// Mitsubishi GX Works2 project: PLC_GROUP_15   PLC: FX3G

// global labels: Global1
VAR_GLOBAL
  Start_Day AT X007 : BOOL;
  End_Day AT M5 : BOOL;
  Work_Day_On AT Y007 : BOOL;
  Input_Raspberry AT D1100 : REAL;
  Input_Lemon AT D1104 : REAL;
  Input_Stabilizer AT D1108 : REAL;
  Input_Gummy AT D1112 : REAL;
  Raspberry_Amount AT D1102 : REAL;
  Lemon_Amount AT D1106 : REAL;
  Stabilizer_Amount AT D1110 : REAL;
  Gummy_Amount AT D1114 : REAL;
  Close_Reset_1 AT CS0 : BOOL;
  Package_Container AT D1126 : REAL;
END_VAR
VAR_GLOBAL CONSTANT
  To_Esroni : REAL := 40;  (* 40 *)
END_VAR
VAR_GLOBAL
  Analog_Output AT D8282 : REAL;
  One_Time_Reset AT CC0 : BOOL;
  Start_Production AT X001 : BOOL;
  Save_Analog_Value AT D8201 : REAL;
END_VAR
VAR_GLOBAL CONSTANT
  CONST400 : REAL := 400;  (* 400 *)
  Min_Regular : REAL;  (* 0 *)
  Max_Regular : REAL := 5;  (* 5 *)
  Min_Pinook : REAL := 6;  (* 6 *)
  Max_Pinook : REAL := 10;  (* 10 *)
END_VAR
VAR_GLOBAL
  Regular AT M3 : BOOL;
  Pinook AT M4 : BOOL;
END_VAR
VAR_GLOBAL CONSTANT
  Check1 : INT := 1;  (* 1 *)
END_VAR
VAR_GLOBAL
  Analog_Input_1 AT D8280 : INT;
  Analog_Real_Value AT D1128 : REAL;
END_VAR
VAR_GLOBAL CONSTANT
  Min_Raspberry_Regular : REAL := 280;  (* 280 *)
  Min_Raspberry_Pinook : REAL := 385;  (* 385 *)
  Min_Lemon_Regular : REAL := 455;  (* 455 *)
  Min_Lemon_Pinook : REAL := 665;  (* 665 *)
  Min_Stabilizer_Regular : REAL := 105;  (* 105 *)
  Min_Stabilizer_Pinook : REAL := 210;  (* 210 *)
  Min_Gummy_Regular : REAL := 28;  (* 28 *)
  Min_Gummy_Pinook : REAL := 70;  (* 70 *)
END_VAR
VAR_GLOBAL
  Check_Product_Raspberry AT M10 : BOOL;
  Check_Product_Lemon AT M20 : BOOL;
  Check_Product_Stabilizer AT M30 : BOOL;
  Check_Product_Gummy AT M40 : BOOL;
  Enough_Products AT M1 : BOOL;
  No_Inventory AT M6 : BOOL;
  Emergency AT X005 : BOOL;
  Timer1 AT TC1 : BOOL;
END_VAR
VAR_GLOBAL CONSTANT
  CONST_5Sec : WORD := 50;  (* 50 *)
END_VAR
VAR_GLOBAL
  Timer_1_Finish AT TS1 : BOOL;
  FiveSecLight AT Y000 : BOOL;
END_VAR
VAR_GLOBAL CONSTANT
  SUB_Res_K280 : REAL := 280;  (* 280 *)
  SUB_Lemon_K455 : REAL := 455;  (* 455 *)
  SUB_Stabi_K105 : REAL := 105;  (* 105 *)
  ADD_Stabi_K35 : REAL := 35;  (* 35 *)
  ADD_Lemon_K455 : REAL := 455;  (* 455 *)
  ADD_Res_K280 : REAL := 280;  (* 280 *)
  ADD_Stabi_K70 : REAL := 70;  (* 70 *)
END_VAR
VAR_GLOBAL
  Raspberry_Cooling_Container AT D1120 : REAL;
  Lemon_Making_Container AT D1118 : REAL;
  Raspberry_Making_Container AT D1116 : REAL;
END_VAR
VAR_GLOBAL CONSTANT
  CONST0 : REAL;  (* 0 *)
  SUB_Res_K385 : REAL := 385;  (* 385 *)
  SUB_Lemon_K665 : REAL := 665;  (* 665 *)
  SUB_Stabi_K210 : REAL := 210;  (* 210 *)
  ADD_Res_K385 : REAL := 385;  (* 385 *)
  ADD_Lemon_K665 : REAL := 665;  (* 665 *)
  ADD_Stabi_K140 : REAL := 140;  (* 140 *)
END_VAR
VAR_GLOBAL
  Can_Start_Cooling AT M21 : BOOL;
  Start_Cooling AT X002 : BOOL;
  Making_finish AT M22 : BOOL;
  Counter_2_finish AT TS2 : BOOL;
  Temperature AT X003 : BOOL;
  CoolingLight AT Y002 : BOOL;
  Timer2 AT TC2 : BOOL;
END_VAR
VAR_GLOBAL CONSTANT
  CONST_8Sec : INT := 80;  (* 80 *)
END_VAR
VAR_GLOBAL
  Lemon_Cooling_Container AT D1122 : REAL;
  Cooling_Finish AT M23 : BOOL;
  Temperature_On AT M24 : BOOL;
END_VAR
VAR_GLOBAL CONSTANT
  SUB_Gummy_K28 : REAL := 28;  (* 28 *)
  SUB_Gummy_K70 : REAL := 70;  (* 70 *)
  ADD_Gummy_K70 : REAL := 70;  (* 70 *)
  ADD_Gummy_K28 : REAL := 28;  (* 28 *)
END_VAR
VAR_GLOBAL
  Mixing_Container AT D1124 : REAL;
  Twinkle_Stop AT M41 : BOOL;
  M_0 AT M0 : BOOL;
  Counter_3_finish AT TS3 : BOOL;
  Timer3 AT TC3 : BOOL;
END_VAR
VAR_GLOBAL CONSTANT
  CONST_1Sec : INT := 10;
END_VAR
VAR_GLOBAL
  Timer4 AT TC4 : BOOL;
  Counter_4_finish AT TS4 : BOOL;  (* 10 *)
  Y_6 AT Y006 : BOOL;
  Y_5 AT Y005 : BOOL;
  Timer5 AT TC5 : BOOL;
END_VAR
VAR_GLOBAL CONSTANT
  Pinook_Blend_Time : INT := 50;  (* 50 *)
  Regular_Blend_Time : INT := 30;  (* 30 *)
END_VAR
VAR_GLOBAL
  Timer6 AT TC6 : BOOL;
  Counter_5_finish AT TS5 : BOOL;
  Counter_6_finish AT TS6 : BOOL;
  Packing_Begin AT M42 : BOOL;
END_VAR
VAR_GLOBAL CONSTANT
  ADD_1_Package : REAL := 1;  (* 1 *)
END_VAR
VAR_GLOBAL
  Cycle_Finished AT M44 : BOOL;
  Timer_3_finish AT TS3 : BOOL;
  Timer_4_finish AT TS4 : BOOL;  (* 10 *)
  Timer_5_finish AT TS5 : BOOL;
  Timer_6_finish AT TS6 : BOOL;
  Timer_2_finish AT TS2 : BOOL;
END_VAR

// task Task_01 (event TRUE, interval 0, priority 31): POU_01

PROGRAM POU_01
(* structured ladder/FBD written out as ST: instructions are called as NAME(EN, inputs, outputs); _pN, _eN, _tN stand for wires *)
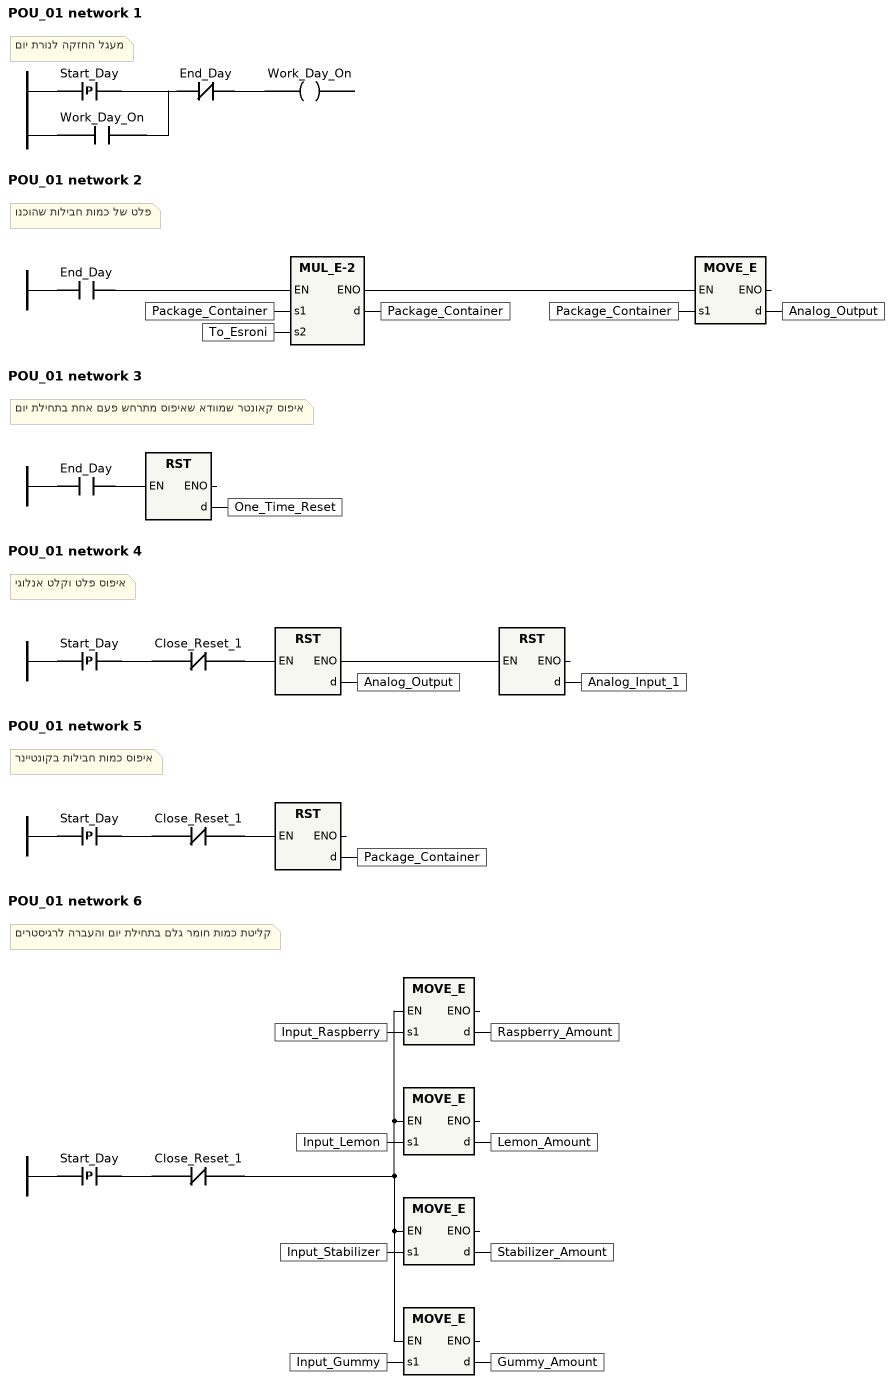
(* network 1 *)
(* מעגל החזקה לנורת יום *)
Work_Day_On := (LDP(TRUE, Start_Day) OR Work_Day_On) AND NOT End_Day;
(* network 2 *)
(* פלט של כמות חבילות שהוכנו *)
_e1 := MUL_E(End_Day, Package_Container, To_Esroni, Package_Container);
MOVE_E(_e1, Package_Container, Analog_Output);
(* network 3 *)
(* איפוס קאונטר שמוודא שאיפוס מתרחש פעם אחת בתחילת יום *)
RST(End_Day, One_Time_Reset);
(* network 4 *)
(* איפוס פלט וקלט אנלוגי *)
_e1 := RST(LDP(TRUE, Start_Day) AND NOT Close_Reset_1, Analog_Output);
RST(_e1, Analog_Input_1);
(* network 5 *)
(* איפוס כמות חבילות בקונטיינר *)
RST(LDP(TRUE, Start_Day) AND NOT Close_Reset_1, Package_Container);
(* network 6 *)
(* קליטת כמות חומר גלם בתחילת יום והעברה לרגיסטרים *)
_p1 := LDP(TRUE, Start_Day) AND NOT Close_Reset_1;
MOVE_E(_p1, Input_Raspberry, Raspberry_Amount);
MOVE_E(_p1, Input_Lemon, Lemon_Amount);
MOVE_E(_p1, Input_Stabilizer, Stabilizer_Amount);
MOVE_E(_p1, Input_Gummy, Gummy_Amount);
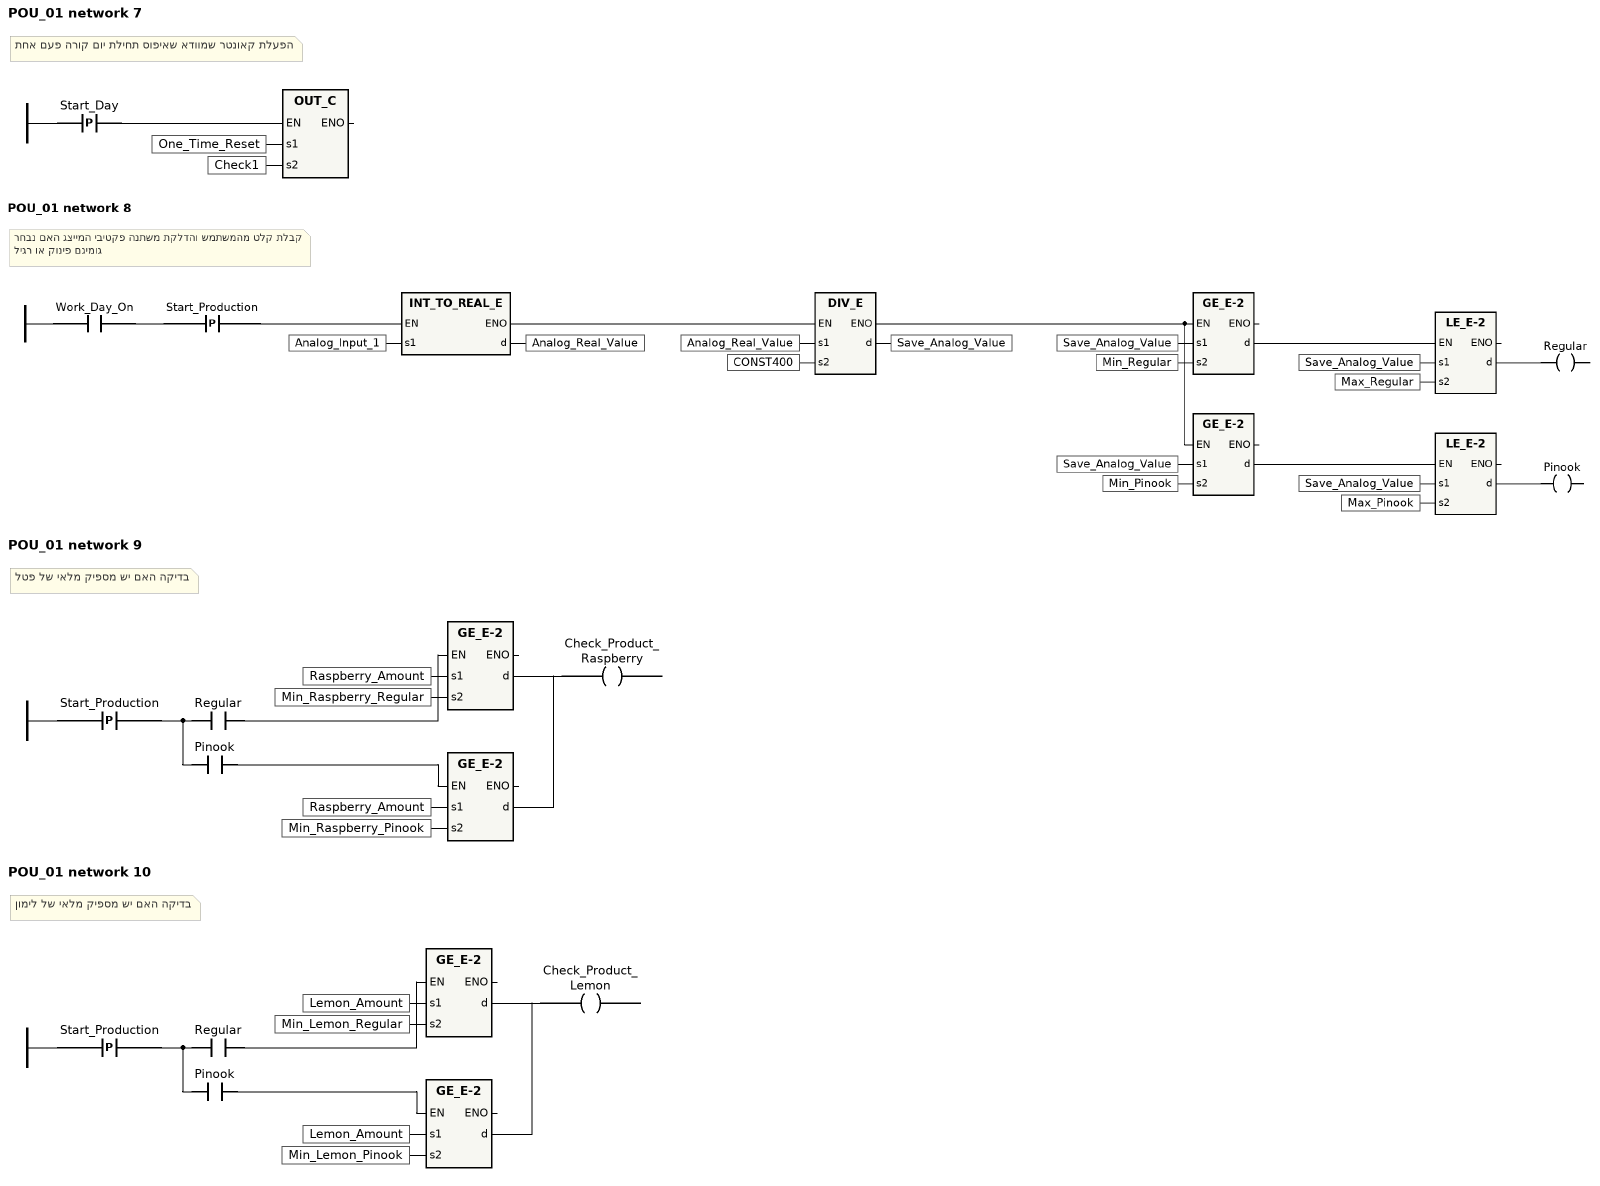
(* network 7 *)
(* הפעלת קאונטר שמוודא שאיפוס תחילת יום קורה פעם אחת *)
OUT_C(LDP(TRUE, Start_Day), One_Time_Reset, Check1);
(* network 8 *)
(* קבלת קלט מהמשתמש והדלקת משתנה פקטיבי המייצג האם נבחר גומיגם פינוק או רגיל *)
_e1 := INT_TO_REAL_E(Work_Day_On AND LDP(TRUE, Start_Production), Analog_Input_1, Analog_Real_Value);
_e2 := DIV_E(_e1, Analog_Real_Value, CONST400, Save_Analog_Value);
GE_E(_e2, Save_Analog_Value, Min_Regular, _t3);
LE_E(_t3, Save_Analog_Value, Max_Regular, _t4);
Regular := _t4;
GE_E(_e2, Save_Analog_Value, Min_Pinook, _t5);
LE_E(_t5, Save_Analog_Value, Max_Pinook, _t6);
Pinook := _t6;
(* network 9 *)
(* בדיקה האם יש מספיק מלאי של פטל *)
_p1 := LDP(TRUE, Start_Production);
GE_E(_p1 AND Regular, Raspberry_Amount, Min_Raspberry_Regular, _t2);
GE_E(_p1 AND Pinook, Raspberry_Amount, Min_Raspberry_Pinook, _t3);
Check_Product_Raspberry := _t2 OR _t3;
(* network 10 *)
(* בדיקה האם יש מספיק מלאי של לימון *)
_p1 := LDP(TRUE, Start_Production);
GE_E(_p1 AND Regular, Lemon_Amount, Min_Lemon_Regular, _t2);
GE_E(_p1 AND Pinook, Lemon_Amount, Min_Lemon_Pinook, _t3);
Check_Product_Lemon := _t2 OR _t3;
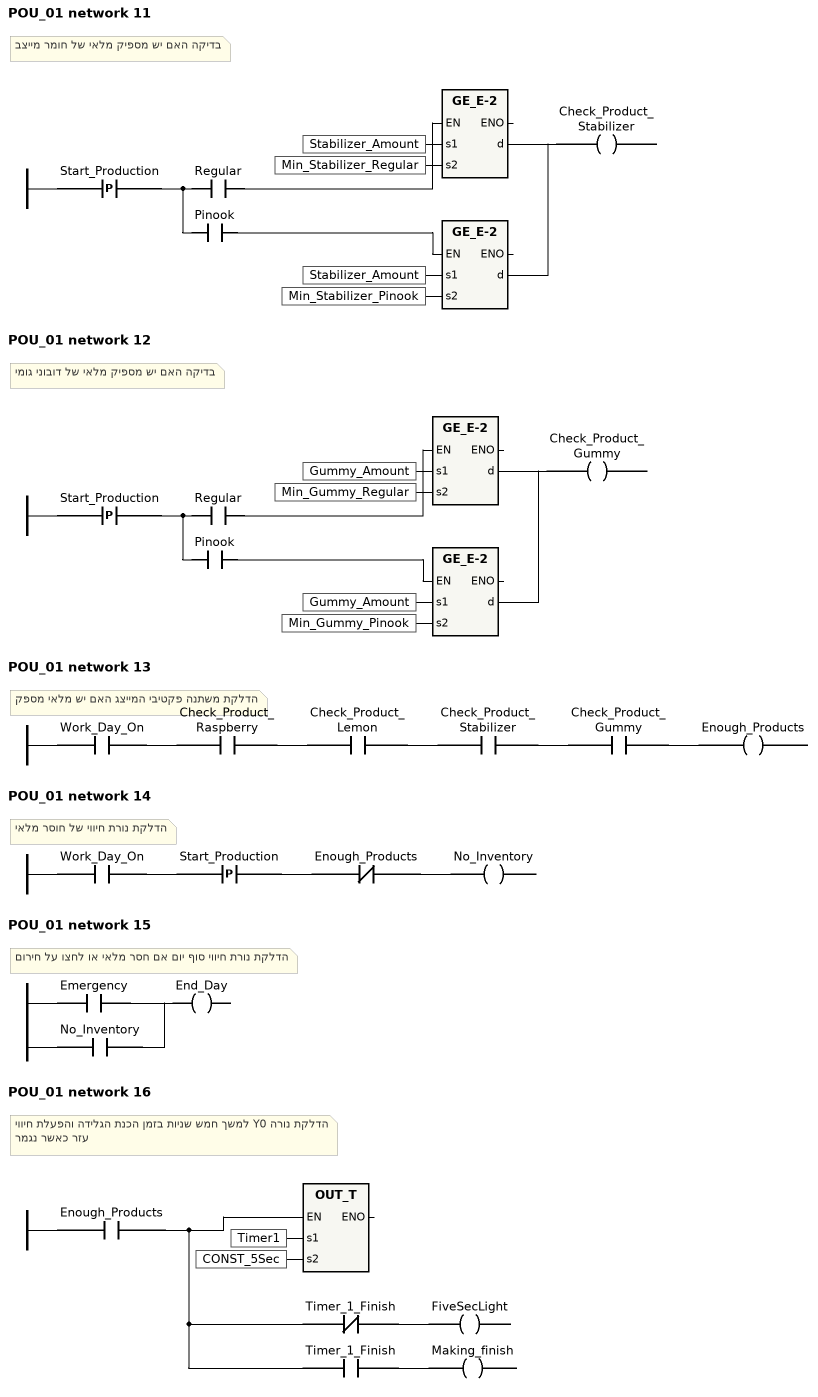
(* network 11 *)
(* בדיקה האם יש מספיק מלאי של חומר מייצב *)
_p1 := LDP(TRUE, Start_Production);
GE_E(_p1 AND Regular, Stabilizer_Amount, Min_Stabilizer_Regular, _t2);
GE_E(_p1 AND Pinook, Stabilizer_Amount, Min_Stabilizer_Pinook, _t3);
Check_Product_Stabilizer := _t2 OR _t3;
(* network 12 *)
(* בדיקה האם יש מספיק מלאי של דובוני גומי *)
_p1 := LDP(TRUE, Start_Production);
GE_E(_p1 AND Regular, Gummy_Amount, Min_Gummy_Regular, _t2);
GE_E(_p1 AND Pinook, Gummy_Amount, Min_Gummy_Pinook, _t3);
Check_Product_Gummy := _t2 OR _t3;
(* network 13 *)
(* הדלקת משתנה פקטיבי המייצג האם יש מלאי מספק *)
Enough_Products := Work_Day_On AND Check_Product_Raspberry AND Check_Product_Lemon AND Check_Product_Stabilizer AND Check_Product_Gummy;
(* network 14 *)
(* הדלקת נורת חיווי של חוסר מלאי *)
No_Inventory := Work_Day_On AND LDP(TRUE, Start_Production) AND NOT Enough_Products;
(* network 15 *)
(* הדלקת נורת חיווי סוף יום אם חסר מלאי או לחצו על חירום *)
End_Day := Emergency OR No_Inventory;
(* network 16 *)
(* הדלקת נורה Y0 למשך חמש שניות בזמן הכנת הגלידה והפעלת חיווי עזר כאשר נגמר *)
FiveSecLight := Enough_Products AND NOT Timer_1_Finish;
OUT_T(Enough_Products, Timer1, CONST_5Sec);
Making_finish := Enough_Products AND Timer_1_Finish;
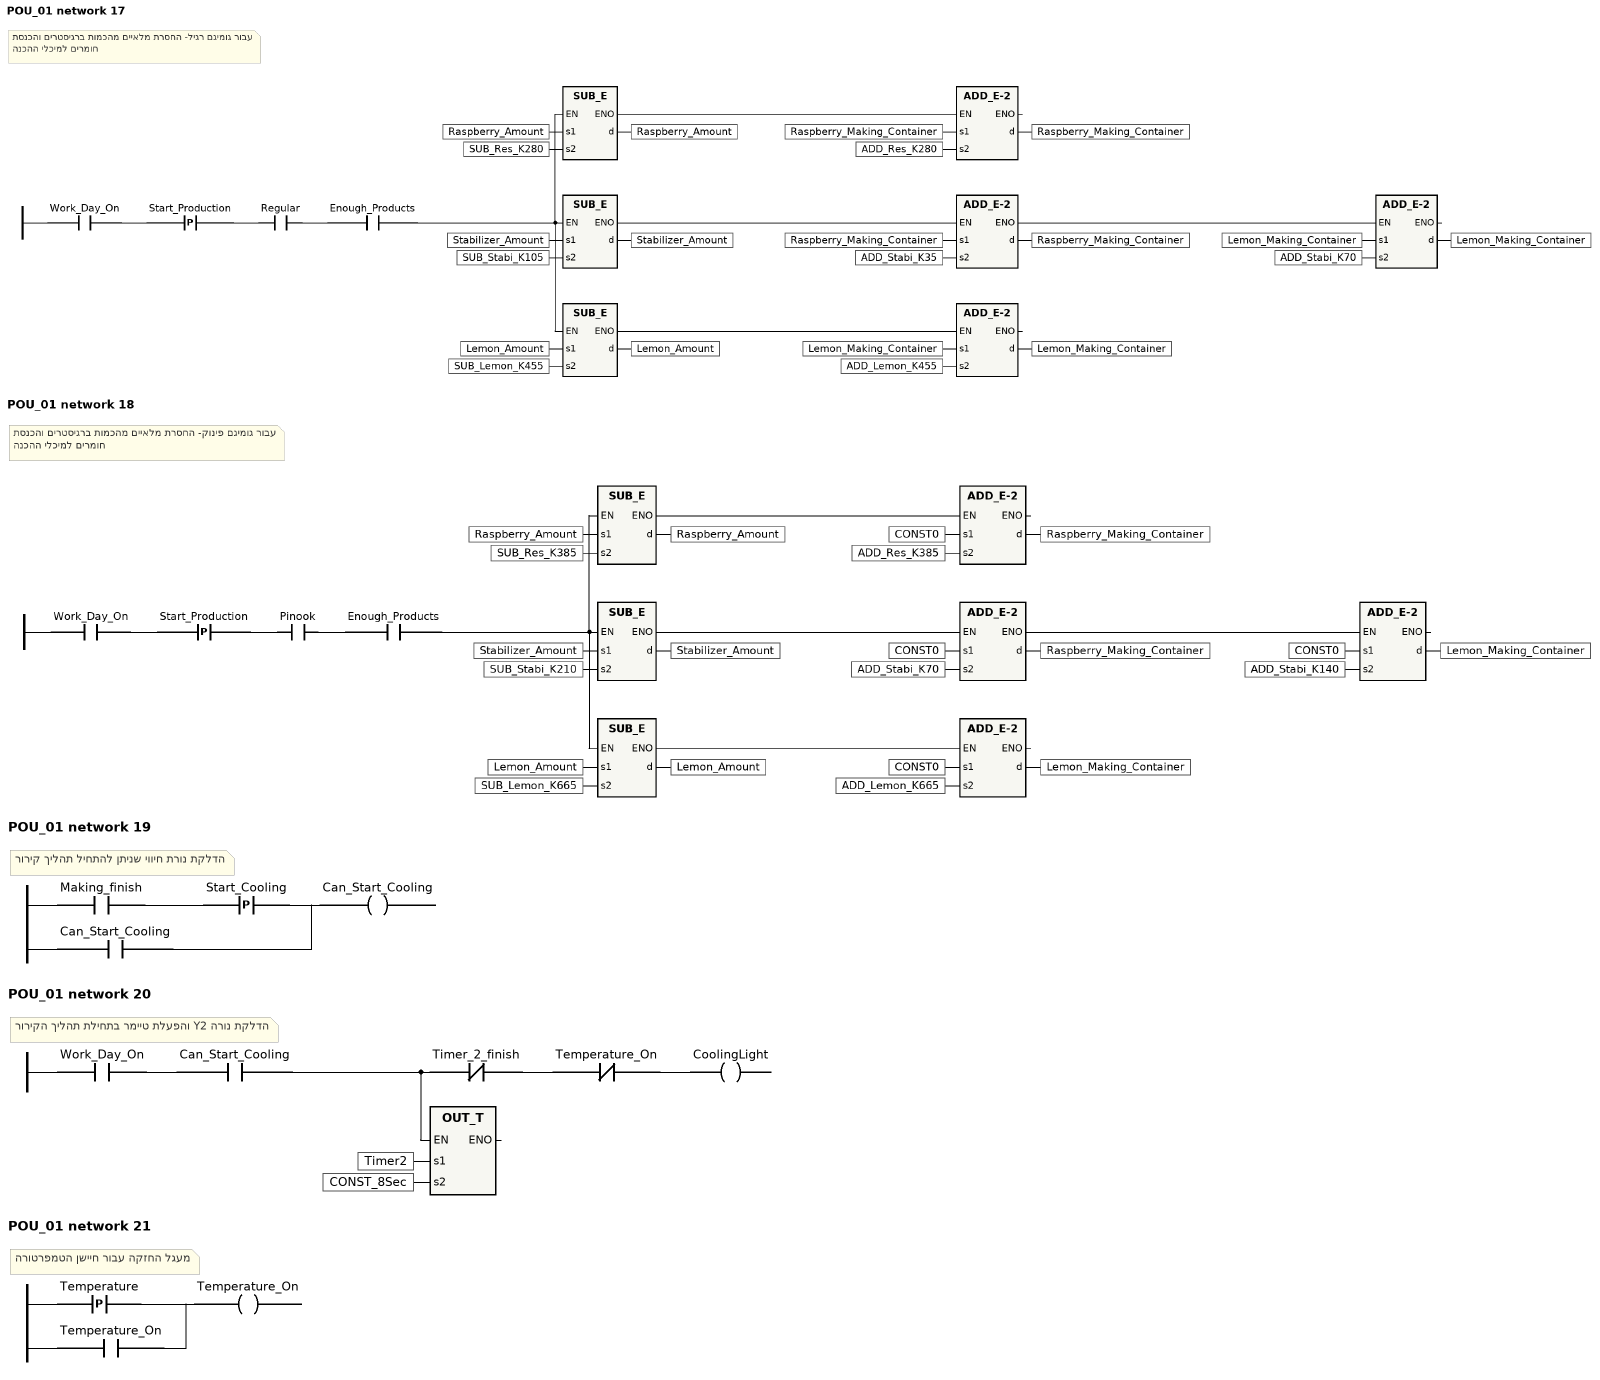
(* network 17 *)
(* עבור גומיגם רגיל- החסרת מלאיים מהכמות ברגיסטרים והכנסת חומרים למיכלי ההכנה *)
_p1 := Work_Day_On AND LDP(TRUE, Start_Production) AND Regular AND Enough_Products;
_e2 := SUB_E(_p1, Raspberry_Amount, SUB_Res_K280, Raspberry_Amount);
ADD_E(_e2, Raspberry_Making_Container, ADD_Res_K280, Raspberry_Making_Container);
_e3 := SUB_E(_p1, Lemon_Amount, SUB_Lemon_K455, Lemon_Amount);
ADD_E(_e3, Lemon_Making_Container, ADD_Lemon_K455, Lemon_Making_Container);
_e4 := SUB_E(_p1, Stabilizer_Amount, SUB_Stabi_K105, Stabilizer_Amount);
_e5 := ADD_E(_e4, Raspberry_Making_Container, ADD_Stabi_K35, Raspberry_Making_Container);
ADD_E(_e5, Lemon_Making_Container, ADD_Stabi_K70, Lemon_Making_Container);
(* network 18 *)
(* עבור גומיגם פינוק- החסרת מלאיים מהכמות ברגיסטרים והכנסת חומרים למיכלי ההכנה *)
_p1 := Work_Day_On AND LDP(TRUE, Start_Production) AND Pinook AND Enough_Products;
_e2 := SUB_E(_p1, Raspberry_Amount, SUB_Res_K385, Raspberry_Amount);
ADD_E(_e2, CONST0, ADD_Res_K385, Raspberry_Making_Container);
_e3 := SUB_E(_p1, Lemon_Amount, SUB_Lemon_K665, Lemon_Amount);
ADD_E(_e3, CONST0, ADD_Lemon_K665, Lemon_Making_Container);
_e4 := SUB_E(_p1, Stabilizer_Amount, SUB_Stabi_K210, Stabilizer_Amount);
_e5 := ADD_E(_e4, CONST0, ADD_Stabi_K70, Raspberry_Making_Container);
ADD_E(_e5, CONST0, ADD_Stabi_K140, Lemon_Making_Container);
(* network 19 *)
(* הדלקת נורת חיווי שניתן להתחיל תהליך קירור *)
Can_Start_Cooling := (Making_finish AND LDP(TRUE, Start_Cooling)) OR Can_Start_Cooling;
(* network 20 *)
(* הדלקת נורה Y2 והפעלת טיימר בתחילת תהליך הקירור *)
_p1 := Work_Day_On AND Can_Start_Cooling;
CoolingLight := _p1 AND NOT Timer_2_finish AND NOT Temperature_On;
OUT_T(_p1, Timer2, CONST_8Sec);
(* network 21 *)
(* מעגל החזקה עבור חיישן הטמפרטורה *)
Temperature_On := LDP(TRUE, Temperature) OR Temperature_On;
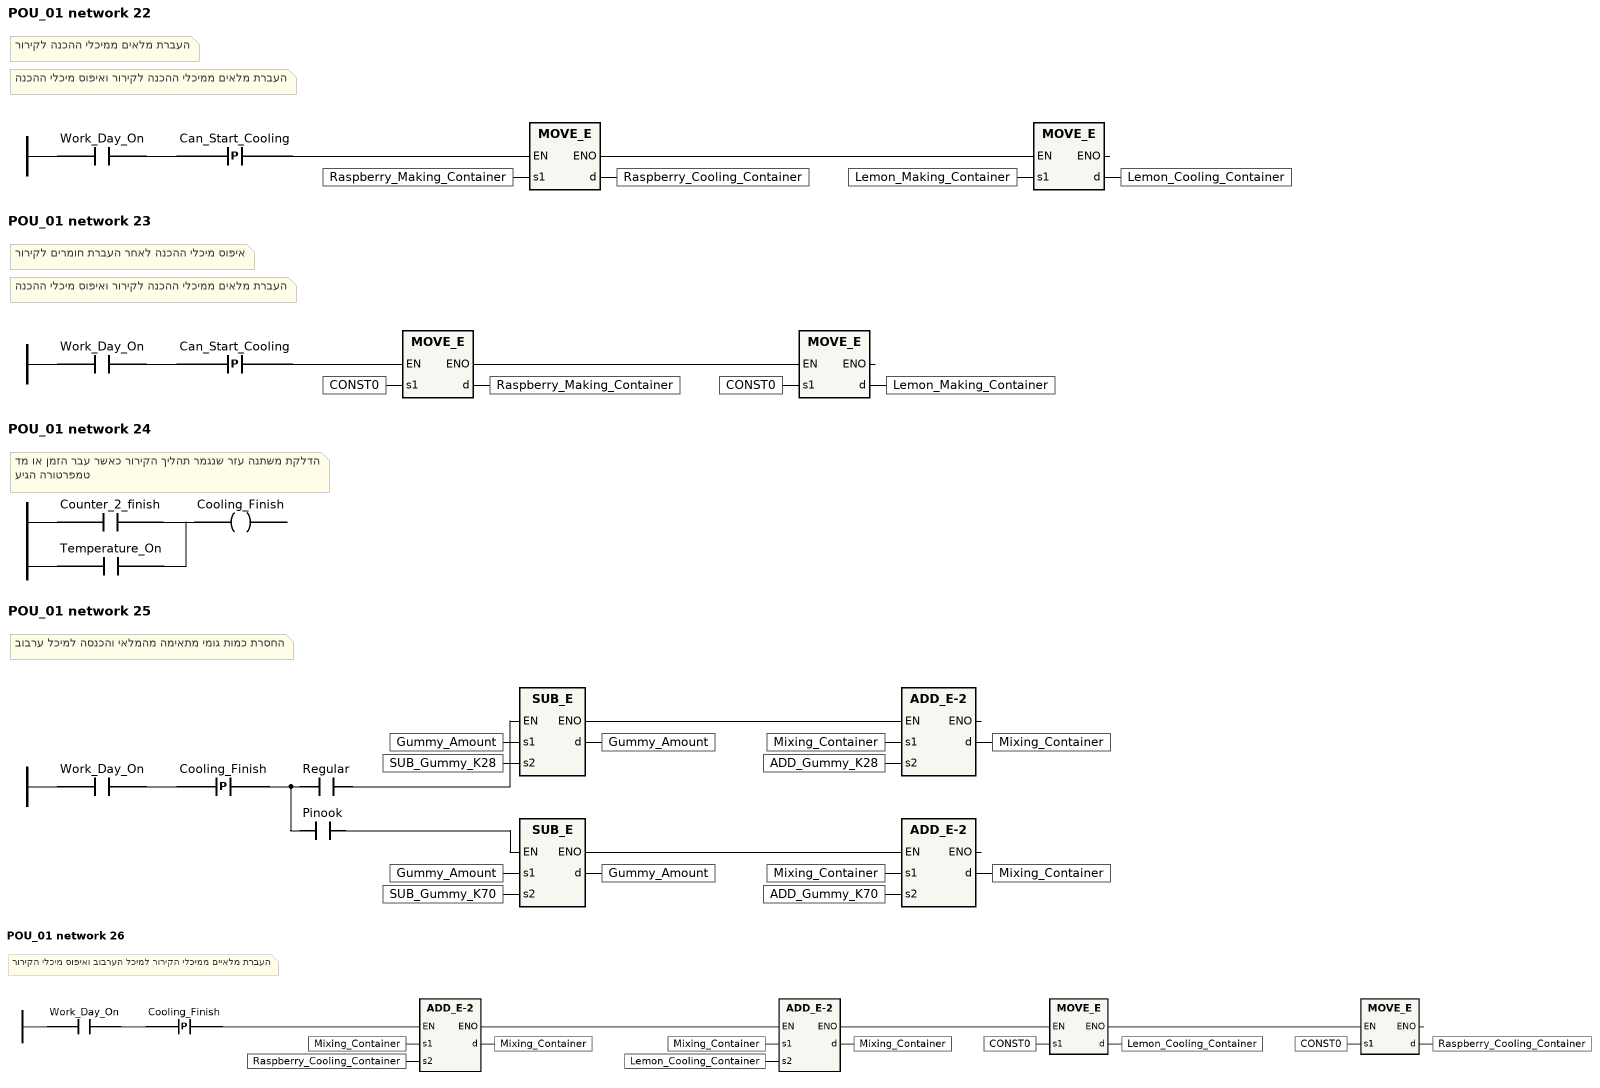
(* network 22 *)
(* העברת מלאים ממיכלי ההכנה לקירור *)
(* העברת מלאים ממיכלי ההכנה לקירור ואיפוס מיכלי ההכנה *)
_e1 := MOVE_E(Work_Day_On AND LDP(TRUE, Can_Start_Cooling), Raspberry_Making_Container, Raspberry_Cooling_Container);
MOVE_E(_e1, Lemon_Making_Container, Lemon_Cooling_Container);
(* network 23 *)
(* איפוס מיכלי ההכנה לאחר העברת חומרים לקירור *)
(* העברת מלאים ממיכלי ההכנה לקירור ואיפוס מיכלי ההכנה *)
_e1 := MOVE_E(Work_Day_On AND LDP(TRUE, Can_Start_Cooling), CONST0, Raspberry_Making_Container);
MOVE_E(_e1, CONST0, Lemon_Making_Container);
(* network 24 *)
(* הדלקת משתנה עזר שנגמר תהליך הקירור כאשר עבר הזמן או מד טמפרטורה הגיע *)
Cooling_Finish := Counter_2_finish OR Temperature_On;
(* network 25 *)
(* החסרת כמות גומי מתאימה מהמלאי והכנסה למיכל ערבוב *)
_p1 := Work_Day_On AND LDP(TRUE, Cooling_Finish);
_e2 := SUB_E(_p1 AND Regular, Gummy_Amount, SUB_Gummy_K28, Gummy_Amount);
ADD_E(_e2, Mixing_Container, ADD_Gummy_K28, Mixing_Container);
_e3 := SUB_E(_p1 AND Pinook, Gummy_Amount, SUB_Gummy_K70, Gummy_Amount);
ADD_E(_e3, Mixing_Container, ADD_Gummy_K70, Mixing_Container);
(* network 26 *)
(* העברת מלאיים ממיכלי הקירור למיכל הערבוב ואיפוס מיכלי הקירור *)
_e1 := ADD_E(Work_Day_On AND LDP(TRUE, Cooling_Finish), Mixing_Container, Raspberry_Cooling_Container, Mixing_Container);
_e2 := ADD_E(_e1, Mixing_Container, Lemon_Cooling_Container, Mixing_Container);
_e3 := MOVE_E(_e2, CONST0, Lemon_Cooling_Container);
MOVE_E(_e3, CONST0, Raspberry_Cooling_Container);
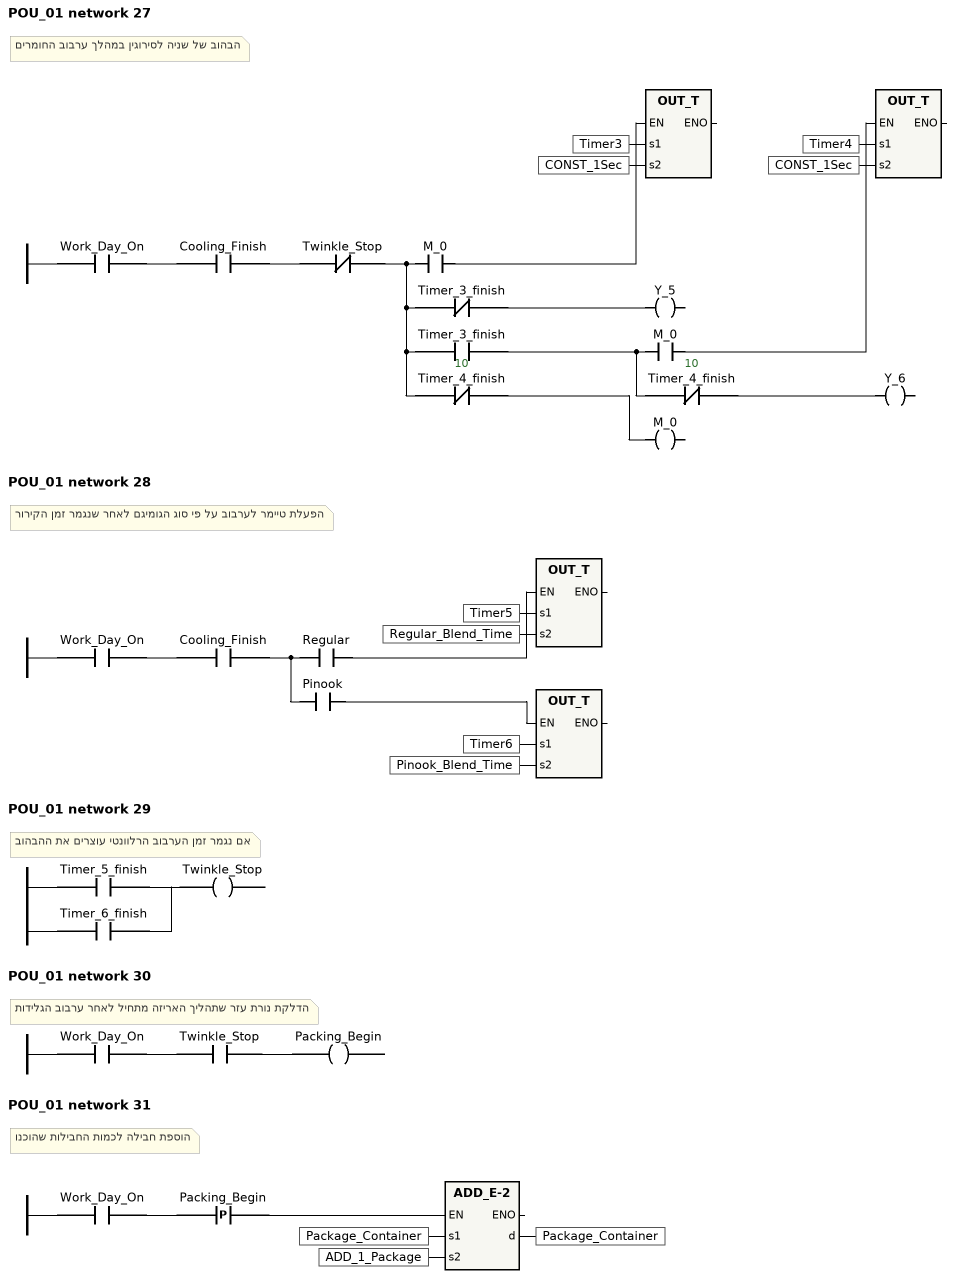
(* network 27 *)
(* הבהוב של שניה לסירוגין במהלך ערבוב החומרים *)
_p1 := Work_Day_On AND Cooling_Finish AND NOT Twinkle_Stop;
OUT_T(_p1 AND M_0, Timer3, CONST_1Sec);
Y_5 := _p1 AND NOT Timer_3_finish;
_p2 := _p1 AND Timer_3_finish;
OUT_T(_p2 AND M_0, Timer4, CONST_1Sec);
Y_6 := _p2 AND NOT Timer_4_finish;
M_0 := _p1 AND NOT Timer_4_finish;
(* network 28 *)
(* הפעלת טיימר לערבוב על פי סוג הגומיגם לאחר שנגמר זמן הקירור *)
_p1 := Work_Day_On AND Cooling_Finish;
OUT_T(_p1 AND Regular, Timer5, Regular_Blend_Time);
OUT_T(_p1 AND Pinook, Timer6, Pinook_Blend_Time);
(* network 29 *)
(* אם נגמר זמן הערבוב הרלוונטי עוצרים את ההבהוב *)
Twinkle_Stop := Timer_5_finish OR Timer_6_finish;
(* network 30 *)
(* הדלקת נורת עזר שתהליך האריזה מתחיל לאחר ערבוב הגלידות *)
Packing_Begin := Work_Day_On AND Twinkle_Stop;
(* network 31 *)
(* הוספת חבילה לכמות החבילות שהוכנו *)
ADD_E(Work_Day_On AND LDP(TRUE, Packing_Begin), Package_Container, ADD_1_Package, Package_Container);
END_PROGRAM
